# EPICS substitutions: depo/depoApp/Db/Neslab_rte.substitutions
file Neslab_rte.template { pattern
{ Sys	, Dev		, PORT		}
{ Depo	, "{Chill:1}"	, Depo_Chill1	}
}
